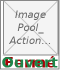
VISUALIZATION Drain  // 60x70
VAR_IN_OUT
	Etat_MaAr	:BOOL;
END_VAR
    Rectangle (0,55 60x15), "Fermé", invisible if: Etat_MaAr, text list: 'OuvFerm', text index: S_Cmd_ElectroValve_Alim_Lavabo
    Rectangle (0,55 60x15), "Ouvert", invisible if: NOT Etat_MaAr, text list: 'OuvFerm', text index: S_Cmd_ElectroValve_Alim_Lavabo
    Image (3,0 55x55), invisible if: Etat_MaAr, image: ImagePool_Action.drain_Close
    Image (3,0 55x55), invisible if: NOT Etat_MaAr, image: ImagePool_Action.drain_Open
END_VISUALIZATION

(* stored: Version 1.1.0.1, ProductVersion 3.1.4024.15
   Visu Drain: Id {96728179-0be9-4287-8f0b-3524cfd737c7} *)
